// TIA Portal V21 export
FUNCTION_BLOCK "PosSenzaDeadBand"   // FB4, LAD
{ S7_Optimized_Access := 'TRUE' }
// stored: MemoryReserve 100, SetENOAutomatically false
   VAR_INPUT
      PosRichiesta : Real;
      PosAttuale : Real;
      ForzaPos : Bool;
      ForzaNeg : Bool;
   END_VAR
   VAR_OUTPUT
      Pos : Bool;
      Neg : Bool;
   END_VAR
   VAR
      DirezioneAvanti : Bool;
      DirezioneIndietro : Bool;
      OldPos : Real;
   END_VAR
BEGIN

REGION Network 1 (SCL)
   IF #OldPos <> #PosRichiesta THEN
       IF #PosAttuale > #PosRichiesta THEN
           #DirezioneAvanti := False;
           #DirezioneIndietro := True;
       ELSE
           #DirezioneAvanti := True;
           #DirezioneIndietro := False;
       END_IF;
       #OldPos :=  #PosRichiesta;
   END_IF;

   IF #DirezioneAvanti AND #PosAttuale >= #PosRichiesta THEN
       #DirezioneAvanti := False;
   END_IF;

   IF #DirezioneIndietro AND #PosAttuale <= #PosRichiesta THEN
       #DirezioneIndietro := False;
   END_IF;

   #Pos := (#DirezioneAvanti OR #ForzaPos) AND NOT #Neg;
   #Neg := (#DirezioneIndietro OR #ForzaNeg) AND NOT #Pos;
END_REGION
END_FUNCTION_BLOCK
